KUKA KRL program: GRUPO1.src

&ACCESS RVP
&REL 81
&PARAM EDITMASK = *
&PARAM TEMPLATE = C:\KRC\Roboter\Template\vorgabe
&PARAM DISKPATH = KRC:\R1\Program\AULA_MEC
DEF GRUPO1( )
;FOLD INI;%{PE}
  ;FOLD USER INI
    ;Make your modifications here

  ;ENDFOLD (USER INI)
;ENDFOLD (INI)
$ADVANCE=0

;FOLD PTP HOME Vel=100 % DEFAULT;%{PE}%R 8.2.24,%MKUKATPBASIS,%CMOVE,%VPTP,%P 1:PTP, 2:HOME, 3:, 5:100, 7:DEFAULT
$BWDSTART=FALSE
PDAT_ACT=PDEFAULT
FDAT_ACT=FHOME
BAS(#PTP_PARAMS,100)
$H_POS=XHOME
PTP XHOME
;ENDFOLD

WRITE10="F"
WRITE5="F"
START_G1="F"

END_G1="F"

PIC_G1="F"





;FOLD LIN P17 Vel=2 m/s CPDAT5 Tool[0] Base[0];%{PE}%R 8.2.24,%MKUKATPBASIS,%CMOVE,%VLIN,%P 1:LIN, 2:P17, 3:, 5:2, 7:CPDAT5
$BWDSTART=FALSE
LDAT_ACT=LCPDAT5
FDAT_ACT=FP17
BAS(#CP_PARAMS,2)
LIN XP17
;ENDFOLD


PIC_G1="T"
LOOP

IF START_G1 == "T" THEN

LIN ENTRY_POINT1

LIN ENTRY_POINT2


LIN ENTRY_POINT3

LIN ENTRY_POINT4


LIN ENTRY_POINT5


WRITE10="T"

LIN ENTRY_POINT6

LIN ENTRY_POINT7


LIN ENTRY_POINT8

LIN ENTRY_POINT9


LIN ENTRY_POINT10


WRITE5="T"



IF END_G1 == "T" THEN

EXIT

ENDIF

ENDIF

ENDLOOP

;FOLD PTP HOME  Vel= 100 % DEFAULT;%{PE}%MKUKATPBASIS,%CMOVE,%VPTP,%P 1:PTP, 2:HOME, 3:, 5:100, 7:DEFAULT
$BWDSTART = FALSE
PDAT_ACT=PDEFAULT
FDAT_ACT=FHOME
BAS (#PTP_PARAMS,100 )
$H_POS=XHOME
PTP  XHOME
;ENDFOLD
END
